// TIA Portal project "Fase3" (V17)

(* hardware
DEVICE "S7-1200 station_1"  S7-1200 Station
   slot 0: "Rack_0"  S7-1200 Rack  Rack  V1.0
   slot 1: "PLC_1"  CPU 1214C AC/DC/Rly  6ES7 214-1BE30-0XB0  V2.2
*)

// ===== PLC "PLC_1"  CPU 1214C AC/DC/Rly =====

VAR_GLOBAL   // PLC tag table "Default tag table"
   "Aumentar" AT %M100.0 : Bool;
   "Disminuir" AT %M100.1 : Bool;
   "Número Total Coches" AT %MW110 : Int;
   "Reset" AT %M120.0 : Bool;
   "Tag_1" AT %MW22 : Word;
   "Tag_2" AT %M125.0 : Bool;
   "Tag_3" AT %M245.0 : Bool;
   "Tag_4" AT %M100.5 : Bool;
   "Tag_5" AT %MW300 : Int;
   "Semaforo Verde" AT %Q0.0 : Bool;
   "Semáforo Amarillo" AT %Q0.1 : Bool;
   "Semáforo Rojo" AT %Q0.2 : Bool;
   "Plazas disponibles" AT %MW0 : Int;
END_VAR

DATA_BLOCK "Contador Ascendente Descendente_DB_1"   // DB1
{ S7_Optimized_Access := 'TRUE' }
VERSION : 0.1
// stored: InstanceOfName Contador Ascendente Descendente
"Contador Ascendente Descendente"
BEGIN
END_DATA_BLOCK

// folder: System blocks/Program resources

DATA_BLOCK "IEC_Counter_0_DB_1"   // DB2
{ S7_Optimized_Access := 'TRUE' }
AUTHOR : Simatic
FAMILY : IEC
NAME : CNTR
VERSION : 1.0
// stored: InstanceOfName IEC_COUNTER
"IEC_COUNTER"
BEGIN
END_DATA_BLOCK

// folder: (top level)

FUNCTION_BLOCK "Contador Ascendente Descendente"   // FB3, LAD
{ S7_Optimized_Access := 'TRUE' }
VERSION : 0.1
   VAR RETAIN
      Num : Int := 100;
   END_VAR
BEGIN

REGION Network 1
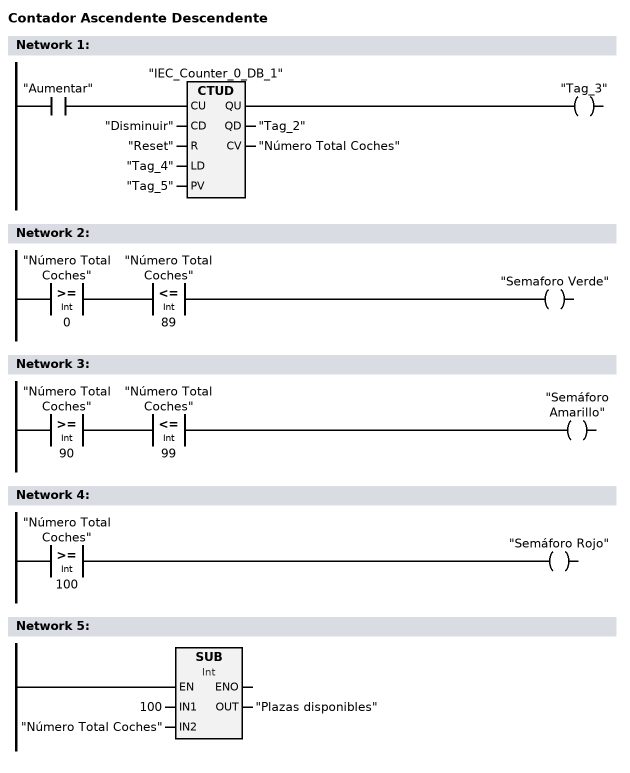
   "IEC_Counter_0_DB_1".CTUD(CU := "Aumentar",
                           CD := "Disminuir",
                           R := "Reset",
                           LD := "Tag_4",
                           PV := "Tag_5",
                           QD => "Tag_2",
                           CV => "Número Total Coches");
   "Tag_3" := "IEC_Counter_0_DB_1".QU;
END_REGION

REGION Network 2
   RUNG wire#powerrail
      { S7_Templates := "SrcType := Int" } GE_Contact(in1 := "Número Total Coches", in2 := 0)
      { S7_Templates := "SrcType := Int" } LE_Contact(in1 := "Número Total Coches", in2 := 89)
      Coil( "Semaforo Verde" )
   END_RUNG
   // the same network as SCL:
   "Semaforo Verde" := ("Número Total Coches" >= 0) AND ("Número Total Coches" <= 89);
END_REGION

REGION Network 3
   RUNG wire#powerrail
      { S7_Templates := "SrcType := Int" } GE_Contact(in1 := "Número Total Coches", in2 := 90)
      { S7_Templates := "SrcType := Int" } LE_Contact(in1 := "Número Total Coches", in2 := 99)
      Coil( "Semáforo Amarillo" )
   END_RUNG
   // the same network as SCL:
   "Semáforo Amarillo" := ("Número Total Coches" >= 90) AND ("Número Total Coches" <= 99);
END_REGION

REGION Network 4
   RUNG wire#powerrail
      { S7_Templates := "SrcType := Int" } GE_Contact(in1 := "Número Total Coches", in2 := 100)
      Coil( "Semáforo Rojo" )
   END_RUNG
   // the same network as SCL:
   "Semáforo Rojo" := "Número Total Coches" >= 100;
END_REGION

REGION Network 5
   RUNG wire#powerrail
      { S7_Templates := "SrcType := Int"; S7_GenerateENO := "TRUE" } Sub(in1 := 100, in2 := "Número Total Coches", out => "Plazas disponibles")
   END_RUNG
   // the same network as SCL:
   "Plazas disponibles" := 100 - "Número Total Coches";
END_REGION
END_FUNCTION_BLOCK

ORGANIZATION_BLOCK "Main"   // OB1, LAD, ProgramCycle
TITLE = "Main Program Sweep (Cycle)"
{ S7_Optimized_Access := 'TRUE' }
VERSION : 0.1
BEGIN

REGION Network 1
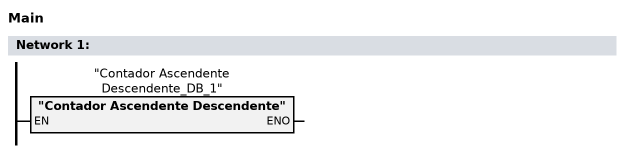
   RUNG wire#powerrail
      "Contador Ascendente Descendente_DB_1"()
   END_RUNG
   // the same network as SCL:
   "Contador Ascendente Descendente_DB_1"();   // "Contador Ascendente Descendente"
END_REGION
END_ORGANIZATION_BLOCK